FUNCTION_BLOCK FB_AnalogOutput
VAR_INPUT
END_VAR
VAR_INPUT
	fValue				: REAL; //input value
END_VAR
VAR_OUTPUT
	nValue 				: INT; //converted value
END_VAR
VAR
	aLimits				: ARRAY[1..2] OF REAL := [0, 100]; //lower and upper limit	
END_VAR

// conversion from Bit value to actual value
nValue := REAL_TO_INT((fValue-aLimits[1])/(aLimits[2]-aLimits[1])*32767);

PROPERTY fLowerLimit : REAL;
GET
fLowerLimit := aLimits[1];
END_GET
SET
aLimits[1] := fLowerLimit;
END_SET
END_PROPERTY

PROPERTY fUpperLimit : REAL;
GET
fUpperLimit := aLimits[2];
END_GET
SET
aLimits[2] := fUpperLimit;
END_SET
END_PROPERTY

END_FUNCTION_BLOCK

(* stored: Version 1.1.0.1, ProductVersion 3.1.4024.9
   POU FB_AnalogOutput: Id {e8cc816e-9340-40fa-8115-6e9fa806b2a4}, SpecialFunc None
   Property fLowerLimit: Id {adb82427-e4b9-4c31-a5bd-ab3e5dd2d104}
   Get Get: Id {ff133f63-b271-4515-87e0-b6d2f7a7b4da}
   Set Set: Id {9c547cbe-dbb5-46b0-81d7-32e2f389816c}
   Property fUpperLimit: Id {e02ae1cb-4796-4557-b671-a31ca10dead6}
   Get Get: Id {bb80768e-2f89-478b-b0f6-c5c862ceefdd}
   Set Set: Id {6741dadc-5f28-4156-aa4b-585c6d01e884} *)
